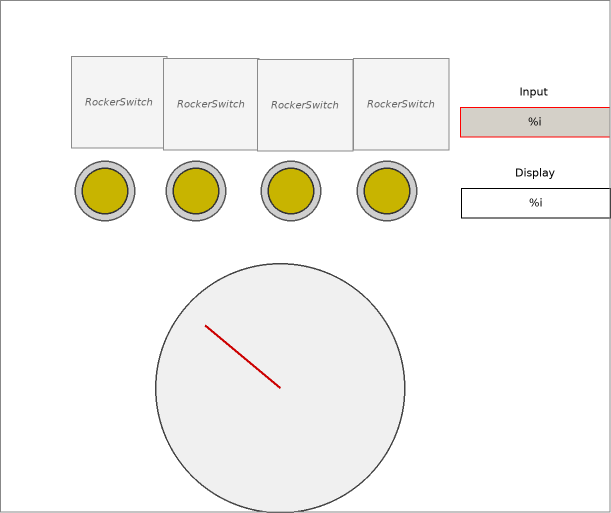
VISUALIZATION Viz1  // 611x513
    Lamp1 (70,156 70x70), variable: IF_Statement.bLight1, style: Lamp-Lamp1-Yellow
    Lamp1 (161,156 70x70), variable: IF_Statement.bLight2, style: Lamp-Lamp1-Yellow
    Lamp1 (256,156 70x70), variable: IF_Statement.bLight3, style: Lamp-Lamp1-Yellow
    Lamp1 (352,156 70x70), variable: IF_Statement.bLight4, style: Lamp-Lamp1-Yellow
    Rectangle (460,107 150x30), "%i", text variable: IF_Statement.iNumber
        OnMouseDown: write the text variable via Default
    Rectangle (461,188 150x30), "%i", text variable: MAIN.iCounterDisp
    Label (459,77 150x30), "Input"
    Label (460,158 150x30), "Display"
    RockerSwitch (71,56 96x92), variable: IF_Statement.bSwitch1, behaviour: TOGGLE, style: Switch-RockerSwitch-Gray
    RockerSwitch (163,58 96x92), variable: IF_Statement.bSwitch2, behaviour: TOGGLE, style: Switch-RockerSwitch-Gray
    RockerSwitch (257,59 96x92), variable: IF_Statement.bSwitch3, behaviour: TOGGLE, style: Switch-RockerSwitch-Gray
    RockerSwitch (353,58 96x92), variable: IF_Statement.bSwitch4, behaviour: TOGGLE, style: Switch-RockerSwitch-Gray
    Meter360 (155,263 250x250), value: IF_Statement.iNumber, style: Meter-Meter360-Gray, scale format: %.1f, scale 0..32000
END_VISUALIZATION

(* stored: Version 1.1.0.1, ProductVersion 3.1.4024.9
   Visu Viz1: Id {b9c525ed-0da0-4195-8f16-01829e78f49b} *)
